{attribute 'qualified_only'}
{attribute 'strict'}
{attribute 'to_string'}
TYPE EventLevel :
(
	INFO := 10,
  WARNING :=20,
  ERROR := 30,
  ALARM := 40
) BYTE := INFO;
END_TYPE

(* stored: Version 1.1.0.1, ProductVersion 3.1.4024.9
   DUT EventLevel: Id {5d6074ed-2b44-44a9-889f-6e1c42bed7e0} *)
